FUNCTION "Message" : Void
{ S7_Optimized_Access := 'TRUE' }
VERSION : 0.1
   VAR_INPUT
      IN_WString : WString;
   END_VAR

   VAR_OUTPUT
      OUT_WString : WString;
   END_VAR

   VAR_IN_OUT
      Cache : "Message_UDT";
   END_VAR


BEGIN
	REGION _name_
	    #OUT_WString := #IN_WString;
	END_REGION







END_FUNCTION

